INTERFACE IProcessSampleMover

METHOD GiveMover : IProcessSampleMover
VAR_INPUT
	mover : REFERENCE TO FB_Mover;
END_VAR
END_METHOD

(* % of completion of the process *)
PROPERTY iCompletionPC : INT
GET
END_GET
END_PROPERTY

(* Process time, expressed in milisecond *)
PROPERTY iProcessTimeMili : DINT
GET
END_GET
SET
END_SET
END_PROPERTY

PROPERTY Mover : REFERENCE TO FB_Mover
GET
END_GET
SET
END_SET
END_PROPERTY

PROPERTY ProcessExecution : ProcessExecution_e
GET
END_GET
SET
END_SET
END_PROPERTY

METHOD TakeMover : IProcessSampleMover
VAR_INPUT
END_VAR
END_METHOD

METHOD ToString : STRING
VAR_INPUT
END_VAR
END_METHOD

PROPERTY xBusy : BOOL
GET
END_GET
SET
END_SET
END_PROPERTY

PROPERTY xDone : BOOL
GET
END_GET
END_PROPERTY

PROPERTY xMoverPathFree : BOOL
GET
END_GET
END_PROPERTY

PROPERTY xMoverShouldLeave : BOOL
GET
END_GET
END_PROPERTY

END_INTERFACE

(* stored: Version 1.1.0.1, ProductVersion 3.1.4024.6
   Itf IProcessSampleMover: Id {195f15bd-9eda-40e2-b294-c2855f6d4080}
   Method GiveMover: Id {05754a6a-14fd-48de-96ed-ce6d8bb38e23}
   Property iCompletionPC: Id {6db509f1-8e66-42c7-a6f6-52dd0036abd7}
   Get Get: Id {bd0f7132-4974-4853-bf43-00fdbbb7be66}
   Property iProcessTimeMili: Id {31e98800-1932-4e20-af14-e98484b89832}
   Get Get: Id {a8082181-d2b9-4efc-a70d-33c8c9c3e426}
   Set Set: Id {a1c93b54-4810-4ec4-b519-5c73fdefb6fb}
   Property Mover: Id {c41497ec-1348-4cbd-95a7-d74ce88b4fa5}
   Get Get: Id {e76e790c-206c-467b-836b-d4f7d9b67b0c}
   Set Set: Id {f5acdb4b-1a0a-41ea-b02d-77cb2e3b4ecf}
   Property ProcessExecution: Id {d6a47de7-07ac-40a7-8905-6b77607cab96}
   Get Get: Id {abfb2323-927a-4eaf-b818-504027a59069}
   Set Set: Id {b50cd2a1-64ca-491a-9967-81f0fe5dab32}
   Method TakeMover: Id {3acae537-92dc-4a43-a882-c4eebcf3abe5}
   Method ToString: Id {05bc73c8-e07f-4c82-97c1-78e00ad73b24}
   Property xBusy: Id {1041503a-54a6-491b-9afa-d4d0ae17ac9e}
   Get Get: Id {3344ece1-021a-4b27-95cb-0b4d6347cdae}
   Set Set: Id {8fcb6030-ecd7-49e6-b79c-3339cfaf6658}
   Property xDone: Id {053db443-2a2e-4ed0-b237-45f4c8234bfc}
   Get Get: Id {927a77db-bfdd-41ad-aa2e-352cdb3b8777}
   Property xMoverPathFree: Id {21f460cf-4be6-4d69-8b42-e843fb9d5832}
   Get Get: Id {2f541f27-218a-4623-bf7e-1e818b56871e}
   Property xMoverShouldLeave: Id {2faa0c16-abad-47e1-b62c-82684c5ff897}
   Get Get: Id {6ea81ec5-f6c7-479b-a111-fb0bb0437553} *)
